ABB RobotStudio station: Versión2.rsstn

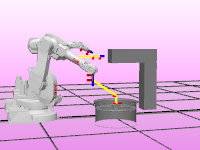
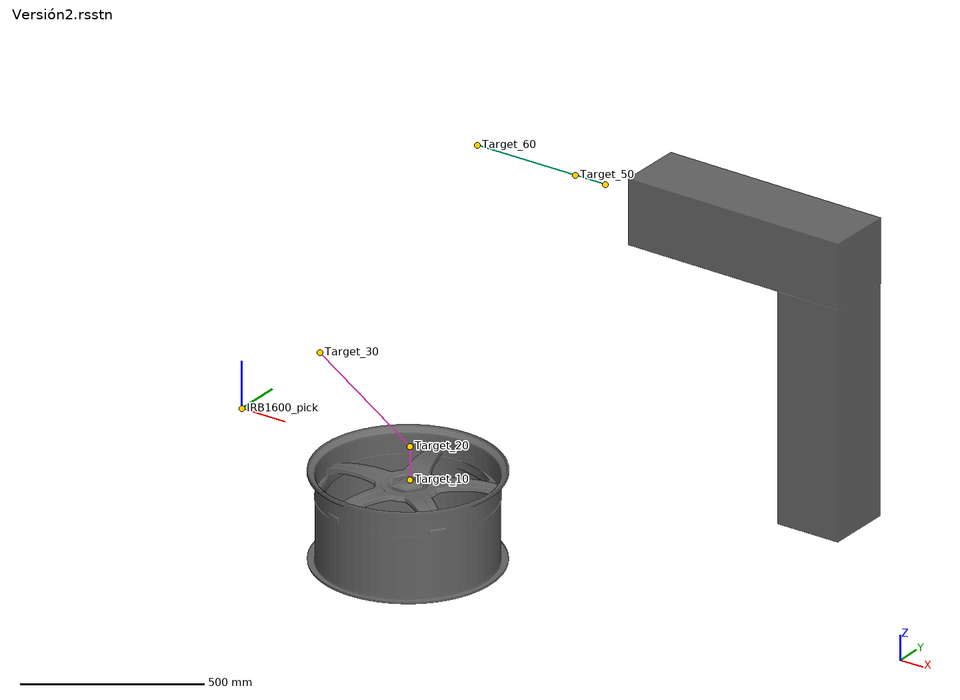
[picture v1: parts stored in the station drawn from their meshes, with robot base, taught points and paths (robot models come from the ABB library and are not in the file)]
Station Versión2 (saved by RobotStudio 21.2.9526.0)
Controller Controlador1
  mechanical unit ROB_1: IRB1600_pick, 6 joints, base frame (0, 0, 0) mm
Layout (positions relative to the parent item):
  - Pieza_8 [part] at (1800, 250, 0) mm, size 200 x 200 x 700 mm
  - base_rueda [part] at (1800, 450, 700) mm, rotated rx 0 ry 0 rz -0.44 deg, size 700 x 200 x 200 mm
  - Smart_Gripper_screw [mechanism, from Tools\ABB_Smart_Gripper_Servo_Fingers.rslib] at (806.29, 800, 929) mm, rotated rx 180 ry 60 rz 180 deg; joint values [0] (rad or m)
  - Rueda [smart component] at (1160, -497.52, 237.67) mm
    - Rueda [part] at (-260, -2.48, -7.41) mm, rotated rx 101.08 ry -90 rz -101.08 deg, size 278.8 x 548.9 x 548.9 mm
  - IRB1600_pick [mechanism, from Robots\IRB1600_6_120_G_02.rslib] at (0, 0, 0) mm; joint values [-0.6874, 0.2303, 0.2671, 0, 1.0734, -0.6874] (rad or m)
  - Mi_Ventosa [smart component, from Downloads\1217c23c-7d3e-48fb-b7d3-d1b2005a3c2bMi_Ventosa.rslib] at (607.28, -498.59, 597.67) mm, rotated rx 180 ry 0 rz -180 deg
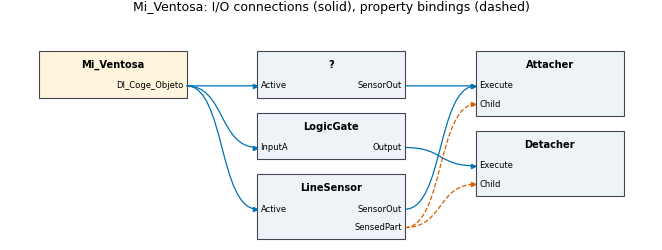
      connections:
        Mi_Ventosa.DI_Coge_Objeto -> ?.Active
        ?.SensorOut -> Attacher.Execute
        Mi_Ventosa.DI_Coge_Objeto -> LogicGate.InputA
        LogicGate.Output -> Detacher.Execute
        Mi_Ventosa.DI_Coge_Objeto -> LineSensor.Active
        LineSensor.SensorOut -> Attacher.Execute
        LineSensor.SensedPart => Attacher.Child
        LineSensor.SensedPart => Detacher.Child
    - Attacher [smart component, from Components\Attacher.rslib]
        properties: Parent=Ventosa; Flange=0; Child=Rueda; Mount=false; Offset=[0 0 0]; Orientation=[0 0 0]
    - Detacher [smart component, from Components\Detacher.rslib]
        properties: Child=Rueda; KeepPosition=true
    - Ventosa [mechanism, from Downloads\1217c23c-7d3e-48fb-b7d3-d1b2005a3c2bMi_Ventosa.rslib] at (0, 0, 0) mm
    - LogicGate [smart component, from Components\LogicGate.rslib]
        properties: Operator=NOT; Delay=0
    - LineSensor [smart component, from Components\LineSensor.rslib]
        properties: Start=[0 0 0.055]; End=[0 0 0.07]; Radius=0.001; SensedPart=Rueda; SensedPoint=[0.907281005859375 -0.498585998535156 0.227922714233398]
      - _sensorPart_ [part]
    - Indicador [part, from Downloads\1217c23c-7d3e-48fb-b7d3-d1b2005a3c2bMi_Ventosa.rslib] at (-4.38, 0, 0) mm
  - IRB1600_screw [mechanism, from Robots\IRB1600_6_120_G_02.rslib] at (0, 800, 0) mm; joint values [0, 0, 0, 0, 0.5236, 0] (rad or m)
Attachment: Mi_Ventosa is attached to IRB1600_pick / Link6
Attachment: Smart_Gripper_screw is attached to IRB1600_screw / Link6
Station logic (signal -> signal, property => property):
  Controlador1.Q_ventosa -> Mi_Ventosa.DI_Coge_Objeto
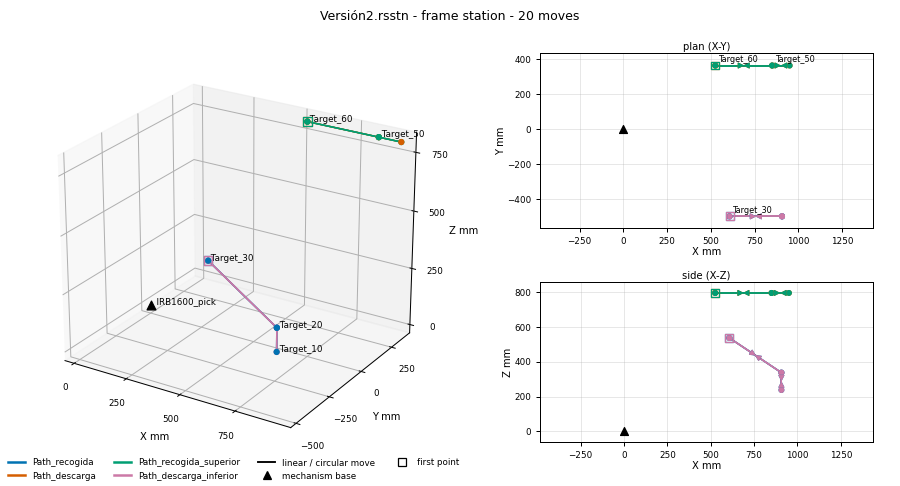
[picture p0: tool path of Versión2.rsstn in frame station, 20 of 20 moves have a stored position in this frame; points joined in program order, loops and branches not executed]
Targets, tools, work objects and paths stored in the station, written as RAPID:
! task T_ROB1
MODULE CalibData
  TASK PERS wobjdata WO_recoger:=[FALSE,TRUE,"",[[906.607,-498.004,237.664],[1,0,0,0]],[[0,0,0],[1,0,0,0]]];
  TASK PERS wobjdata WO_descargar:=[FALSE,TRUE,"",[[1038.626,-225.1,0],[1,0,0,0]],[[0,0,0],[1,0,0,0]]];
  PERS tooldata TCP_Ventosa:=[TRUE,[[0,0,60],[1,0,0,0]],[0.1,[0,0,1],[1,0,0,0],0,0,0]];
ENDMODULE

! task T_ROB1
MODULE Module1
  CONST robtarget Target_10:=[[0.674,-0.582,0.001],[0,0,1,0],[0,0,0,0],[9E+09,9E+09,9E+09,9E+09,9E+09,9E+09]];
  CONST robtarget Target_20:=[[0.674,-0.582,100.001],[0,0,1,0],[-1,0,-1,0],[9E+09,9E+09,9E+09,9E+09,9E+09,9E+09]];
  CONST robtarget Target_30:=[[-299.326,-0.582,300.001],[0,0,1,0],[-1,0,-1,0],[9E+09,9E+09,9E+09,9E+09,9E+09,9E+09]];
  CONST robtarget Target_40:=[[-87.95,588.826,797.258],[0.707106781,0,0.707106781,0],[0,-2,1,0],[9E+09,9E+09,9E+09,9E+09,9E+09,9E+09]];
  CONST robtarget Target_50:=[[-187.95,588.826,797.258],[0.707106781,0,0.707106781,0],[0,-2,1,0],[9E+09,9E+09,9E+09,9E+09,9E+09,9E+09]];
  CONST robtarget Target_60:=[[-512.95,588.826,797.258],[0.707106781,0,0.707106781,0],[0,-2,1,0],[9E+09,9E+09,9E+09,9E+09,9E+09,9E+09]];
  PROC Path_recogida()
    MoveJ Target_30,v500,z0,TCP_Ventosa\WObj:=WO_recoger;
    MoveL Target_20,v500,z0,TCP_Ventosa\WObj:=WO_recoger;
    MoveL Target_10,v500,z0,TCP_Ventosa\WObj:=WO_recoger;
    SetDO Q_ventosa,1;
    WaitTime 1;
    MoveL Target_20,v500,z0,TCP_Ventosa\WObj:=WO_recoger;
    MoveL Target_30,v500,z0,TCP_Ventosa\WObj:=WO_recoger;
  ENDPROC
  PROC main()
    Path_recogida;
    Path_descarga;
    Path_recogida_superior;
    Path_descarga_inferior;
  ENDPROC
  PROC Path_descarga()
    MoveJ Target_60,v500,z0,TCP_Ventosa\WObj:=WO_descargar;
    MoveL Target_50,v500,z0,TCP_Ventosa\WObj:=WO_descargar;
    MoveL Target_40,v500,z0,TCP_Ventosa\WObj:=WO_descargar;
    WaitTime 1;
    MoveL Target_50,v500,z0,TCP_Ventosa\WObj:=WO_descargar;
    SetDO Q_ventosa,0;
    MoveL Target_60,v500,z0,TCP_Ventosa\WObj:=WO_descargar;
  ENDPROC
  PROC Path_recogida_superior()
    MoveJ Target_60,v500,z0,TCP_Ventosa\WObj:=WO_descargar;
    MoveL Target_50,v500,z0,TCP_Ventosa\WObj:=WO_descargar;
    MoveL Target_40,v500,z0,TCP_Ventosa\WObj:=WO_descargar;
    SetDO Q_ventosa,1;
    WaitTime 1;
    MoveL Target_50,v500,z0,TCP_Ventosa\WObj:=WO_descargar;
    MoveL Target_60,v500,z0,TCP_Ventosa\WObj:=WO_descargar;
  ENDPROC
  PROC Path_descarga_inferior()
    MoveJ Target_30,v500,z0,TCP_Ventosa\WObj:=WO_recoger;
    MoveL Target_20,v500,z0,TCP_Ventosa\WObj:=WO_recoger;
    MoveL Target_10,v500,z0,TCP_Ventosa\WObj:=WO_recoger;
    WaitTime 1;
    MoveL Target_20,v500,z0,TCP_Ventosa\WObj:=WO_recoger;
    SetDO Q_ventosa,0;
    MoveL Target_30,v500,z0,TCP_Ventosa\WObj:=WO_recoger;
  ENDPROC
ENDMODULE

! task (no controller)
MODULE CalibData
  PERS tooldata Servo:=[TRUE,[[0,0,114.2],[1,0,0,0]],[0.215,[8.7,12.3,49.2],[1,0,0,0],0.00021,0.00024,0.00009]];
ENDMODULE

